SUBAPPLICATION Uebung_072 (* GBSD auf UT ausgeben *)
  (* Standard: 61499-2 *)
  (* Version 1.0, 2023-10-23, franz *)
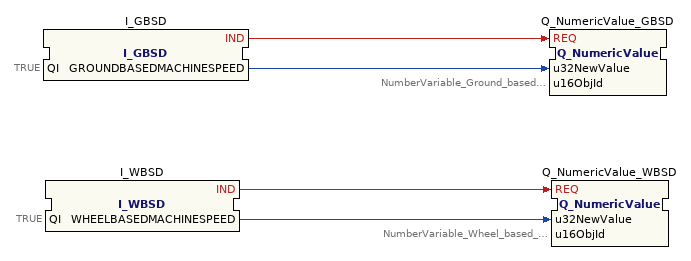
  FBS
    I_GBSD : I_GBSD(QI := TRUE);
    Q_NumericValue_GBSD : Q_NumericValue(u16ObjId := NumberVariable_Ground_based_machine_speed);
    I_WBSD : I_WBSD(QI := TRUE);
    Q_NumericValue_WBSD : Q_NumericValue(u16ObjId := NumberVariable_Wheel_based_machine_speed);
  END_FBS
  EVENT_CONNECTIONS
    I_GBSD.IND TO Q_NumericValue_GBSD.REQ;
    I_WBSD.IND TO Q_NumericValue_WBSD.REQ;
  END_CONNECTIONS
  DATA_CONNECTIONS
    I_GBSD.GROUNDBASEDMACHINESPEED TO Q_NumericValue_GBSD.u32NewValue;
    I_WBSD.WHEELBASEDMACHINESPEED TO Q_NumericValue_WBSD.u32NewValue;
  END_CONNECTIONS
END_SUBAPPLICATION
